// LS Electric XG5000 project: 2023-09-05 #1
// PLC NewPLC
// module base 0 slot 0: 입출력 모듈:XBC-DR32H (DC 24V 입력, 릴레이 출력 32점)

PROGRAM NewProgram (task: 스캔 프로그램)

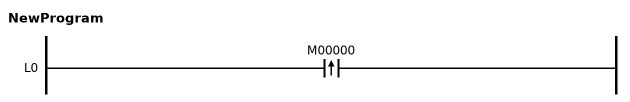
; L0
LOADP     M00000

VARIABLES AND COMMENTS (devices not used above)
P00000	BIT	PB1
P00020	BIT	PL1